{attribute 'qualified_only' := ''}
{attribute 'strict' := ''}
TYPE MOTION_STATUS :
(
	ConstantVelocity := 0,
	Accelerating := 1,
	Decelerating := 2
);
END_TYPE

(* stored: Version 1.1.0.1, ProductVersion 3.1.4024.11
   DUT MOTION_STATUS: Id {d0691f08-49ad-48b3-80f9-43631fa4594b} *)
